VAR_GLOBAL
	arAxisCtrl_gb : ARRAY[1..uiMAX_AXIS_INDEX] OF Axis_Ctrl_gb;
	arAxisStutus_gb : ARRAY[1..uiMAX_AXIS_INDEX] OF Axis_Status_gb;
END_VAR

(* stored: Version 1.1.0.1, ProductVersion 3.1.4024.11
   GVL Global_Axis_Interface: Id {dacf9f9d-d6b8-4d74-913a-d6d76ed6e141} *)
